// TIA Portal V17 export
// export: Created 2022-07-06T15:40:15.3080344Z, ExportSetting WithDefaults, DisplayName Totally Integrated Automation Portal, DisplayVersion V17, DisplayName TIA Portal Openness, DisplayVersion V17, DisplayName TIA Portal Teamcenter Gateway, DisplayVersion V17, DisplayName TIA Portal Version Control Interface, DisplayVersion V17, DisplayName SINAMICS Startdrive Advanced, DisplayVersion V17, DisplayName SINAMICS Startdrive G130, G150, S120, S150, SINAMICS MV, S210, DisplayVersion V17, DisplayName SINAMICS Startdrive G110M, G120, G120C, G120D, G120P, G115D, DisplayVersion V17, DisplayName STEP 7 Professional, DisplayVersion V17, DisplayName STEP 7 Safety, DisplayVersion V17, DisplayName WinCC Advanced / Unified PC, DisplayVersion V17
FUNCTION_BLOCK "Block_1TEST_2"   // FB1, LAD
{ S7_Optimized_Access := 'TRUE' }
VERSION : 0.1
// stored: AutoNumber true, IsIECCheckEnabled false, IsRetainMemResEnabled false, MemoryReserve 100, SetENOAutomatically false, UDAEnableTagReadback false
   VAR_INPUT
      "test entrée" : Bool;
   END_VAR
   VAR_OUTPUT
      "test sortie" : Bool;
   END_VAR
BEGIN

REGION Network 1
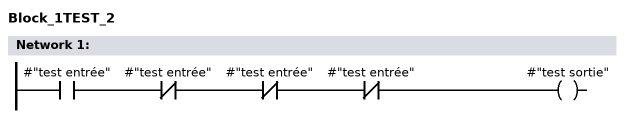
   RUNG wire#powerrail
      Contact( #"test entrée" )
      I_Contact( #"test entrée" )
      I_Contact( #"test entrée" )
      I_Contact( #"test entrée" )
      Coil( #"test sortie" )
   END_RUNG
   // the same network as SCL:
   #"test sortie" := #"test entrée" AND NOT #"test entrée" AND NOT #"test entrée" AND NOT #"test entrée";
END_REGION
END_FUNCTION_BLOCK
